PROGRAM RETURN_FUKUDA_1
VAR
END_VAR

CASE INPUT_VAR.I_CASE OF
0:
	IF INPUT_VAR.ACTIVE_ID=6 THEN
		INPUT_VAR.ACTIVE_ID:=1;
	END_IF
//	FUKUDA_MOVE(STEP_DATA_1:=0,STEP_DATA_2:=0,STEP_DATA_3:=0,STEP_DATA_4:=0,STEP_DATA_5:=2);
	CASE INPUT_VAR.I_CURRENT_TRANSACTION.TRANSPORT_INDEX OF
		2 : FUKUDA_MOVE(STEP_DATA_1:=3,
				STEP_DATA_2:=0,
				STEP_DATA_3:=3,
				STEP_DATA_4:=0,//2, //2
				STEP_DATA_5:=1);

		1 : FUKUDA_MOVE(STEP_DATA_1:=3,
				STEP_DATA_2:=0,
				STEP_DATA_3:=3,
				STEP_DATA_4:=1,//2, //2
				STEP_DATA_5:=0);
	END_CASE
1:
	IF INPUT_VAR.ACTIVE_ID=6 THEN
		INPUT_VAR.ACTIVE_ID:=1;
	END_IF
	
//	FUKUDA_MOVE(STEP_DATA_1:=6,STEP_DATA_2:=1,STEP_DATA_3:=21,STEP_DATA_4:=0,STEP_DATA_5:=0);
	FUKUDA_MOVE(STEP_DATA_1:=3,
				STEP_DATA_2:=0,
				STEP_DATA_3:=3,
				STEP_DATA_4:=0,
				STEP_DATA_5:=0);

2:
	IF INPUT_VAR.ACTIVE_ID=6 THEN
		INPUT_VAR.ACTIVE_ID:=1;
	END_IF
	
//	FUKUDA_MOVE(STEP_DATA_1:=6,STEP_DATA_2:=1,STEP_DATA_3:=21,STEP_DATA_4:=0,STEP_DATA_5:=0);
	FUKUDA_MOVE(STEP_DATA_1:=3,
				STEP_DATA_2:=0,
				STEP_DATA_3:=3,
				STEP_DATA_4:=0,
				STEP_DATA_5:=0);

3:
	IF INPUT_VAR.ACTIVE_ID=6 THEN
		INPUT_VAR.ACTIVE_ID:=1;
	END_IF
	
//	FUKUDA_MOVE(STEP_DATA_1:=6,STEP_DATA_2:=2,STEP_DATA_3:=21,STEP_DATA_4:=0,STEP_DATA_5:=0);
	FUKUDA_MOVE(STEP_DATA_1:=INPUT_VAR.I_CURRENT_TRANSACTION.TRANSPORT_INDEX+4,
				STEP_DATA_2:=1,
				STEP_DATA_3:=21,
				STEP_DATA_4:=0,
				STEP_DATA_5:=0);

4:
	IF INPUT_VAR.ACTIVE_ID=6 THEN
		INPUT_VAR.ACTIVE_ID:=1;
	END_IF
	
//	FUKUDA_MOVE(STEP_DATA_1:=6,STEP_DATA_2:=2,STEP_DATA_3:=21,STEP_DATA_4:=0,STEP_DATA_5:=0);
	FUKUDA_MOVE(STEP_DATA_1:=INPUT_VAR.I_CURRENT_TRANSACTION.TRANSPORT_INDEX+4,
				STEP_DATA_2:=1,
				STEP_DATA_3:=21,
				STEP_DATA_4:=0,
				STEP_DATA_5:=0);

5:
	IF INPUT_VAR.ACTIVE_ID=6 THEN
		INPUT_VAR.ACTIVE_ID:=1;
	END_IF
	
//	FUKUDA_MOVE(STEP_DATA_1:=6,STEP_DATA_2:=2,STEP_DATA_3:=21,STEP_DATA_4:=0,STEP_DATA_5:=0);
	FUKUDA_MOVE(STEP_DATA_1:=INPUT_VAR.I_CURRENT_TRANSACTION.TRANSPORT_INDEX+4,
				STEP_DATA_2:=2,
				STEP_DATA_3:=21,
				STEP_DATA_4:=0,
				STEP_DATA_5:=);
6:
	IF INPUT_VAR.ACTIVE_ID=6 THEN
		INPUT_VAR.ACTIVE_ID:=1;
	END_IF
	
//	FUKUDA_MOVE(STEP_DATA_1:=6,STEP_DATA_2:=2,STEP_DATA_3:=21,STEP_DATA_4:=0,STEP_DATA_5:=0);
	FUKUDA_MOVE(STEP_DATA_1:=INPUT_VAR.I_CURRENT_TRANSACTION.TRANSPORT_INDEX+4,
				STEP_DATA_2:=2,
				STEP_DATA_3:=2,
				STEP_DATA_4:=0,
				STEP_DATA_5:=0);
	input_var.o_CARTESSIAN_GRIPPER_ON:=TRUE;
	input_var.o_CARTESSIAN_GRIPPER_Off:=FALSE;
7:
	IF INPUT_VAR.ACTIVE_ID=6 THEN
		INPUT_VAR.ACTIVE_ID:=1;
	END_IF
	
	//	FUKUDA_MOVE(STEP_DATA_1:=1,STEP_DATA_2:=2,STEP_DATA_3:=3,STEP_DATA_4:=0,STEP_DATA_5:=0);
	FUKUDA_MOVE(STEP_DATA_1:=INPUT_VAR.I_CURRENT_TRANSACTION.STATION_NUMBER_LOAD,
				STEP_DATA_2:=2,
				STEP_DATA_3:=INPUT_VAR.I_CURRENT_TRANSACTION.JIG_INDEX_LOAD+4,
				STEP_DATA_4:=0,
				STEP_DATA_5:=0);

8:
	IF INPUT_VAR.ACTIVE_ID=6 THEN
		INPUT_VAR.ACTIVE_ID:=1;
	END_IF
//	FUKUDA_MOVE(STEP_DATA_1:=1,STEP_DATA_2:=4,STEP_DATA_3:=13,STEP_DATA_4:=0,STEP_DATA_5:=0);
	FUKUDA_MOVE(STEP_DATA_1:=INPUT_VAR.I_CURRENT_TRANSACTION.STATION_NUMBER_LOAD,
				STEP_DATA_2:=3,
				STEP_DATA_3:=INPUT_VAR.I_CURRENT_TRANSACTION.JIG_INDEX_LOAD+10,
				STEP_DATA_4:=0,
				STEP_DATA_5:=0);

9: 
	IF INPUT_VAR.ACTIVE_ID=6 THEN
		INPUT_VAR.ACTIVE_ID:=1;
	END_IF
	
//	FUKUDA_MOVE(STEP_DATA_1:=1,STEP_DATA_2:=3,STEP_DATA_3:=3,STEP_DATA_4:=0,STEP_DATA_5:=0);
	FUKUDA_MOVE(STEP_DATA_1:=INPUT_VAR.I_CURRENT_TRANSACTION.STATION_NUMBER_LOAD,
				STEP_DATA_2:=3,
				STEP_DATA_3:=INPUT_VAR.I_CURRENT_TRANSACTION.JIG_INDEX_LOAD+10,
				STEP_DATA_4:=0,
				STEP_DATA_5:=0);
10: 
	IF INPUT_VAR.ACTIVE_ID=6 THEN
		INPUT_VAR.ACTIVE_ID:=1;
	END_IF
	
//	FUKUDA_MOVE(STEP_DATA_1:=1,STEP_DATA_2:=3,STEP_DATA_3:=3,STEP_DATA_4:=0,STEP_DATA_5:=0);
	FUKUDA_MOVE(STEP_DATA_1:=INPUT_VAR.I_CURRENT_TRANSACTION.STATION_NUMBER_LOAD,
				STEP_DATA_2:=3,
				STEP_DATA_3:=INPUT_VAR.I_CURRENT_TRANSACTION.JIG_INDEX_LOAD+10,
				STEP_DATA_4:=0,
				STEP_DATA_5:=0);
11:
	IF INPUT_VAR.ACTIVE_ID=6 THEN
		INPUT_VAR.ACTIVE_ID:=1;
	END_IF
//	FUKUDA_MOVE(STEP_DATA_1:=1,STEP_DATA_2:=3,STEP_DATA_3:=13,STEP_DATA_4:=0,STEP_DATA_5:=0);
	FUKUDA_MOVE(STEP_DATA_1:=INPUT_VAR.I_CURRENT_TRANSACTION.STATION_NUMBER_LOAD,
				STEP_DATA_2:=4,
				STEP_DATA_3:=INPUT_VAR.I_CURRENT_TRANSACTION.JIG_INDEX_LOAD,
				STEP_DATA_4:=0,
				STEP_DATA_5:=0);

	input_var.o_CARTESSIAN_GRIPPER_ON:=FALSE;
	input_var.o_CARTESSIAN_GRIPPER_Off:=TRUE;
12: 
	
	IF INPUT_VAR.ACTIVE_ID=6 THEN
		INPUT_VAR.ACTIVE_ID:=1;
	END_IF
//	FUKUDA_MOVE(STEP_DATA_1:=1,STEP_DATA_2:=4,STEP_DATA_3:=3,STEP_DATA_4:=0,STEP_DATA_5:=0);
	FUKUDA_MOVE(STEP_DATA_1:=INPUT_VAR.I_CURRENT_TRANSACTION.STATION_NUMBER_LOAD,
				STEP_DATA_2:=3,
				STEP_DATA_3:=INPUT_VAR.I_CURRENT_TRANSACTION.JIG_INDEX_LOAD,
				STEP_DATA_4:=0,
				STEP_DATA_5:=0);
13: 
	
	IF INPUT_VAR.ACTIVE_ID=6 THEN
		INPUT_VAR.ACTIVE_ID:=1;
	END_IF
//	FUKUDA_MOVE(STEP_DATA_1:=1,STEP_DATA_2:=4,STEP_DATA_3:=3,STEP_DATA_4:=0,STEP_DATA_5:=0);
	FUKUDA_MOVE(STEP_DATA_1:=INPUT_VAR.I_CURRENT_TRANSACTION.STATION_NUMBER_LOAD,
				STEP_DATA_2:=3,
				STEP_DATA_3:=INPUT_VAR.I_CURRENT_TRANSACTION.JIG_INDEX_LOAD,
				STEP_DATA_4:=0,
				STEP_DATA_5:=0);

14: 
	
	IF INPUT_VAR.ACTIVE_ID=6 THEN
		INPUT_VAR.ACTIVE_ID:=1;
	END_IF
//	FUKUDA_MOVE(STEP_DATA_1:=1,STEP_DATA_2:=4,STEP_DATA_3:=3,STEP_DATA_4:=0,STEP_DATA_5:=0);
	FUKUDA_MOVE(STEP_DATA_1:=INPUT_VAR.I_CURRENT_TRANSACTION.STATION_NUMBER_LOAD,
				STEP_DATA_2:=4,
				STEP_DATA_3:=INPUT_VAR.I_CURRENT_TRANSACTION.JIG_INDEX_LOAD,
				STEP_DATA_4:=0,
				STEP_DATA_5:=0);

15:
	
	IF INPUT_VAR.ACTIVE_ID=6 THEN
		INPUT_VAR.ACTIVE_ID:=1;
	END_IF
	
//	FUKUDA_MOVE(STEP_DATA_1:=0,STEP_DATA_2:=1,STEP_DATA_3:=0,STEP_DATA_4:=0,STEP_DATA_5:=0);
	FUKUDA_MOVE(STEP_DATA_1:=0,
				STEP_DATA_2:=1,
				STEP_DATA_3:=0,
				STEP_DATA_4:=0,
				STEP_DATA_5:=0);

	END_CASE

END_PROGRAM

(* stored: Version 1.1.0.1, ProductVersion 3.1.4020.12
   POU RETURN_FUKUDA_1: Id {6883359e-21d5-424a-b6e6-733132b757c2}, SpecialFunc None *)
